FUNCTION_BLOCK BfbOneWayCtrl
  (* Standard: 61499-2 *)
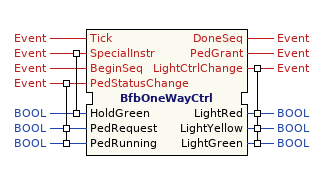
  EVENT_INPUT
    Tick;
    SpecialInstr WITH HoldGreen;
    BeginSeq;
    PedStatusChange WITH PedRequest, PedRunning;
  END_EVENT
  EVENT_OUTPUT
    DoneSeq;
    PedGrant;
    LightCtrlChange WITH LightRed, LightYellow, LightGreen;
  END_EVENT
  VAR_INPUT
    HoldGreen : BOOL := 0;
    PedRequest : BOOL := 0;
    PedRunning : BOOL := 0;
  END_VAR
  VAR_OUTPUT
    LightRed : BOOL := 0;
    LightYellow : BOOL := 0;
    LightGreen : BOOL := 0;
  END_VAR
  VAR
    d : UDINT := 0;
    greenTicks : UDINT := 15000000;
    yellowTicks : UDINT := 5000000;
    redTicks : UDINT := 2000000;
  END_VAR
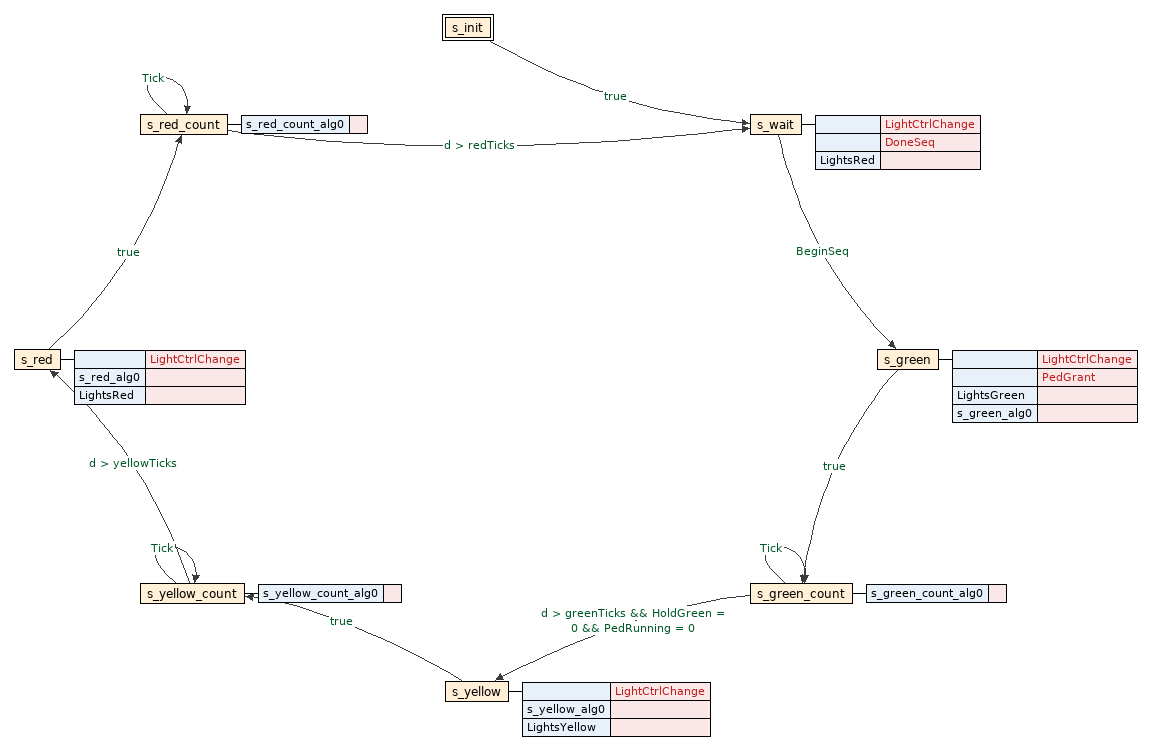
  EC_STATES
    s_init;
    s_wait : -> LightCtrlChange, -> DoneSeq, LightsRed;
    s_green : -> LightCtrlChange, -> PedGrant, LightsGreen, s_green_alg0;
    s_green_count : s_green_count_alg0;
    s_yellow : -> LightCtrlChange, s_yellow_alg0, LightsYellow;
    s_yellow_count : s_yellow_count_alg0;
    s_red : -> LightCtrlChange, s_red_alg0, LightsRed;
    s_red_count : s_red_count_alg0;
  END_STATES
  EC_TRANSITIONS
    s_init TO s_wait := true;
    s_wait TO s_green := BeginSeq;
    s_green TO s_green_count := true;
    s_green_count TO s_yellow := d > greenTicks && HoldGreen = 0 && PedRunning = 0;
    s_green_count TO s_green_count := Tick;
    s_yellow TO s_yellow_count := true;
    s_yellow_count TO s_red := d > yellowTicks;
    s_yellow_count TO s_yellow_count := Tick;
    s_red TO s_red_count := true;
    s_red_count TO s_wait := d > redTicks;
    s_red_count TO s_red_count := Tick;
  END_TRANSITIONS
  ALGORITHM s_green_alg0 IN ST:
d := 0;
  END_ALGORITHM
  ALGORITHM s_green_count_alg0 IN ST:
if d <= greenTicks then d := d + 1; end_if;
  END_ALGORITHM
  ALGORITHM s_yellow_alg0 IN ST:
d := 0;
  END_ALGORITHM
  ALGORITHM s_yellow_count_alg0 IN ST:
d := d + 1;
  END_ALGORITHM
  ALGORITHM s_red_alg0 IN ST:
d := 0;
  END_ALGORITHM
  ALGORITHM s_red_count_alg0 IN ST:
d := d + 1;
  END_ALGORITHM
  ALGORITHM LightsRed IN ST:
        LightRed := 1;
        LightYellow := 0;
        LightGreen := 0;
  END_ALGORITHM
  ALGORITHM LightsYellow IN ST:
        LightRed := 0;
        LightYellow := 1;
        LightGreen := 0;
  END_ALGORITHM
  ALGORITHM LightsGreen IN ST:
        LightRed := 0;
        LightYellow := 0;
        LightGreen := 1;
  END_ALGORITHM
END_FUNCTION_BLOCK
